FUNCTION_BLOCK Mc2MoveModuloTask EXTENDS Mc2MotionTask
VAR
	_TargetPosition : LREAL;
	_Direction		: Tc2_MC2.MC_Direction;
	McMoveModulo	: ARRAY[0..1] OF Tc2_MC2.MC_MoveModulo;
	Active			: UDINT;
    _McBufferMode	: Tc2_MC2.MC_BufferMode;
	_MoveOptions	: Tc2_MC2.ST_MoveOptions;
END_VAR

PROPERTY BufferMode : REFERENCE TO MC_BufferMode
GET
BufferMode REF= _McBufferMode;
END_GET
END_PROPERTY

{attribute 'monitoring' := 'call'}
PROPERTY Busy : BOOL
GET
Busy := McMoveModulo[Active].Busy;
END_GET
END_PROPERTY

METHOD CyclicLogic
VAR
    i : UDINT;
END_VAR
FOR i := 0 TO 1 DO
    McMoveModulo[i](Axis		  := _Axis.Axis,
                    Position	  := _TargetPosition,
                    Direction	  := _Direction,
                    Velocity	  := _Axis.Velocity,
                    Acceleration := _Axis.Acceleration,
                    Deceleration := _Axis.Deceleration,
                    Jerk		  := _Axis.Jerk,
                    BufferMode	  := _McBufferMode,
                    Options	  := _MoveOptions);
    
    McMoveModulo[i].Execute := FALSE;
END_FOR
END_METHOD

PROPERTY Direction : MC_Direction
SET
_Direction := Direction;
END_SET
END_PROPERTY

{attribute 'monitoring' := 'call'}
PROPERTY Error : BOOL
GET
Error := McMoveModulo[Active].Error;
END_GET
END_PROPERTY

{attribute 'monitoring' := 'call'}
PROPERTY ErrorId : UDINT
GET
ErrorID := McMoveModulo[Active].ErrorID;
END_GET
END_PROPERTY

METHOD Execute : BOOL;
IF Active = 0 THEN
	Active := 1;
	McMoveModulo[Active](Axis		  := _Axis.Axis,
						 Execute	  := TRUE,
						 Position	  := _TargetPosition,
						 Direction	  := _Direction,
						 Velocity	  := _Axis.Velocity,
						 Acceleration := _Axis.Acceleration,
						 Deceleration := _Axis.Deceleration,
						 Jerk		  := _Axis.Jerk,
						 BufferMode	  := _McBufferMode,
						 Options	  := _MoveOptions);
ELSE
	Active := 0;
	McMoveModulo[Active](Axis		  := _Axis.Axis,
						 Execute	  := TRUE,
						 Position	  := _TargetPosition,
						 Direction	  := _Direction,
						 Velocity	  := _Axis.Velocity,
						 Acceleration := _Axis.Acceleration,
						 Deceleration := _Axis.Deceleration,
						 Jerk		  := _Axis.Jerk,
						 BufferMode	  := _McBufferMode,
						 Options	  := _MoveOptions);
END_IF

Execute := TRUE;
END_METHOD

PROPERTY MoveOptions : REFERENCE TO ST_MoveOptions
GET
MoveOptions REF= _MoveOptions;
END_GET
END_PROPERTY

{attribute 'monitoring' := 'call'}
PROPERTY TargetPosition : LREAL
SET
_TargetPosition := TargetPosition;
END_SET
END_PROPERTY

END_FUNCTION_BLOCK

(* stored: Version 1.1.0.1, ProductVersion 3.1.4026.20
   POU Mc2MoveModuloTask: Id {498b828b-fecf-4de3-8779-49001f9deaea}, SpecialFunc None
   Property BufferMode: Id {bc106bac-6533-42fe-8929-0582f9fa6340}
   Get Get: Id {05d97c69-6ddc-4821-86ba-e0e6b76c6cf2}
   Property Busy: Id {9dac919a-303b-4478-a5d9-5d51b21e7038}
   Get Get: Id {3eede686-e5ed-468e-93db-f6f1cf2bc254}
   Method CyclicLogic: Id {1ab634e9-e5e8-4361-aefb-53a4d29daae0}
   Property Direction: Id {803ecd2e-14fd-4570-b166-79f035cfd335}
   Set Set: Id {4636ff88-35d7-4287-be8f-2024276f07f7}
   Property Error: Id {34ab9a64-cdc1-4edb-ac5f-a1171bdab3c9}
   Get Get: Id {3b8b4c4c-3633-4e11-83bf-ac5909581096}
   Property ErrorId: Id {7d6c9fb4-f1eb-4848-8ed7-37ab5b79b6a3}
   Get Get: Id {8b9db3ca-c086-4473-916d-3fd744cfedfd}
   Method Execute: Id {515a7d5e-031d-4721-b407-8f2103a448b6}
   Property MoveOptions: Id {02a55eeb-d353-4af9-8ad8-d9033bd3cd98}
   Get Get: Id {012df2dc-61c8-4ea5-a775-e36b9d036936}
   Property TargetPosition: Id {b70d736f-6e4f-4075-9f07-03367a17ef37}
   Set Set: Id {efe7885d-bfd6-4042-a44b-45779d17c4c3} *)
